Staubli VAL3: LasMAN.pjx

--- LasMAN.pjx ---
Parameters version=s7.7 stackSize=10000 millimeterUnit=true
Program file=Main.pgx
Program file=OnEvent1.pgx
Program file=OnEvent10.pgx
Program file=OnEvent11.pgx
Program file=OnEvent12.pgx
Program file=OnEvent13.pgx
Program file=OnEvent14.pgx
Program file=OnEvent15.pgx
Program file=OnEvent16.pgx
Program file=OnEvent17.pgx
Program file=OnEvent18.pgx
Program file=OnEvent19.pgx
Program file=OnEvent2.pgx
Program file=OnEvent3.pgx
Program file=OnEvent4.pgx
Program file=OnEvent5.pgx
Program file=OnEvent6.pgx
Program file=OnEvent7.pgx
Program file=OnEvent8.pgx
Program file=OnEvent9.pgx
Program file=Welcome.pgx
Program file=start.pgx
Program file=stop.pgx
Data file=LasMAN.dtx
Library alias=TxtFile path=Disk://TxtFile/TxtFile.pjx autoload=true password=
Library alias=UI path=Disk://StaubliUI/StaubliUI.pjx autoload=true password=
Library alias=DataBase path=Disk://DataBase/DataBase.pjx autoload=true password=
Library alias=Kit path=Disk://Kit/Kit.pjx autoload=true password=
Library alias=Teach path=Disk://Teach/Teach.pjx autoload=true password=
Library alias=IO path=Disk://IO/IO.pjx autoload=true password=
Library alias=ExtAxis path=Disk://extAxisCan/extAxisCan.pjx autoload=false password=

--- LasMAN.dtx ---
bool bExit
bool bSync
bool bWelcome = true

--- Main.pgx ---
program Main()
  local num l_nKey
begin

  //-----------------------------------------------------------------------
  //Header begin
  //Description of program
  //  根据不同类型的报警和当前机器人所处的运行状态处理报警事件
  //Input parameters
  //
  //Output paramaters
  //Example
  //  call Main()
  //History
  //  Creation : 2013-06-23
  //Header end
  //-----------------------------------------------------------------------
  //主程序


  //等按钮松开
  wait(getKey()==-1)
  do
    //每个操作模式之前的动作
    cls()
    userPage()
    resetMotion()
    call UI:Control_PanelMd("请等待，正在载入库......")


    //
    switch DataBase:nInterfaceType
      case 1
        //手动回零
        call OnEvent1()
      break
      case 2
        //手动对齐
        call OnEvent2()
      break
      case 3
        //编辑工艺
        call OnEvent3()
      break
      case 4
        //编辑动作
        call OnEvent4()
      break
      case 5
        //编辑产品
        call OnEvent5()
      break
      case 6
        //远程
        call OnEvent6()
      break
      //选项
      case 7
        call OnEvent7()
      break
      case 8
        //退出
        call OnEvent8()
      break
      case 9
        //主界面
        call OnEvent9()
      break
      case 10
        //示教产品的用户坐标系
        call OnEvent10()
      break

      case 11
        //示教产品偏差
        call OnEvent11()
      break

      //异步第七轴
      case 12
        call OnEvent12()
      break

      //生产
      case 13
        call OnEvent13()
      break


      //示教工具
      case 14
        call OnEvent14()
      break


      //示教Home
      case 15
        call OnEvent15()
      break


      //异步第八轴
      case 16
        call OnEvent16()
      break


      //替换空白调试文件
      case 17
        call OnEvent17()
      break


      //示教同步七轴
      case 18
        call OnEvent18()
      break

      //示教同步八轴
      case 19
        call OnEvent19()
      break


      //其他非法标志符，则退出
      default
        bExit=true
      break

    endSwitch

    delay(0)
  until bExit
  //Exit
  call stop()

end

--- start.pgx ---
program start()
  local bool l_bRes
begin

  //-----------------------------------------------------------------------
  //Header begin
  //Description of program
  //  LasMAN启动程序
  //Input parameters
  //
  //Output paramaters
  //
  //Creation : 2013.10.22 Ye yanjie  y.ye@staubli.com
  //Header end
  //-----------------------------------------------------------------------
  logMsg("运行lasman")
  DataBase:sSoftWareTime="2015_02_03"
  setTextMode(0)
  $jogPage(false)
  bWelcome=false
  taskCreate "Welcom",100,Welcome()



  //获取机器版本
  DataBase:sVersion[0]=getVersion("System")
  DataBase:sVersion[1]=getVersion("ArmType")
  DataBase:sVersion[2]=getVersion("Mounting")
  DataBase:sVersion[3]=getVersion("ControllerSN")
  DataBase:nRemoteProduct=0



  //删除备份
  $delete("Disk://BackUp")
  $delete("Disk://OffTxt")

  //参数初始化
  disablePower()
  bExit=false
  DataBase:nProductCount=0
  DataBase:bSaveTrajPoint=false
  TxtFile:tCfg.trsf=TxtFile:tFileTool.trsf={0,0,0,0,0,0}
  TxtFile:trPointCount={0,0,0,0,0,0}
  resetMotion()
  //设置默认的boxcar为0，10
  $setBoxcarFreq(0,10)


  //检查相应的文件是否正确
  call TxtFile:IsFileOK(l_bRes)
  if !l_bRes
    bWelcome=true
    delay(0)
    // popUpMsg("文本文件不正确!")
    call stop()
    return
  endIf

  //IO初始化
  call IO:Init()
  DataBase:nInterfaceType=9


  //外部轴初始化
  call Kit:ExtraSysAxisIni(l_bRes)
  if !l_bRes
    return
  endIf




  //建立新的进程
  taskCreate "LasMan",100,Main()
  taskCreate "Poll",100,Kit:Poll()
  bWelcome=true

end

--- OnEvent1.pgx ---
program OnEvent1()
  local bool l_bRes
begin
  //-----------------------------------------------------------------------
  //Header begin
  //LasMAN3.6
  //Description of program
  //
  //Input parameters
  //
  //Output paramaters
  //Example
  //  call OnEvent1()
  //History
  //  Creation : 2013-06-23  y.ye@staubli.com
  //Header end
  //-----------------------------------------------------------------------

  DataBase:bStopPoll=true
  call TxtFile:ReadCfg(l_bRes)
  IO:bWeldEnable=TxtFile:bWeldEnable
  IO:bWeldEnable=TxtFile:bWeldEnable
  IO:bExt7AxisEnable=TxtFile:b7Axis
  IO:bExt8AxisEnable=TxtFile:b8Axis
  DataBase:bStopPoll=false

  if l_bRes

    call Kit:GoHome()
  else
    popUpMsg("读取配置文件出错")
  endIf
  DataBase:nInterfaceType=9
end

--- OnEvent10.pgx ---
program OnEvent10()
begin
  //-----------------------------------------------------------------------
  //Header begin
  //LasMAN3.6
  //Description of program
  //
  //Input parameters
  //
  //Output paramaters
  //Example
  //  call OnEvent1()
  //History
  //  Creation : 2013-06-23  y.ye@staubli.com
  //Header end
  //-----------------------------------------------------------------------
  resetMotion()
  call Teach:TeachFrame(DataBase:fFrame)
  DataBase:nInterfaceType=9
end

--- OnEvent11.pgx ---
program OnEvent11()
begin
  //-----------------------------------------------------------------------
  //Header begin
  //LasMAN3.6
  //Description of program
  //
  //Input parameters
  //
  //Output paramaters
  //Example
  //  call OnEvent1()
  //History
  //  Creation : 2013-06-23  y.ye@staubli.com
  //Header end
  //-----------------------------------------------------------------------
  //示教偏差
  resetMotion()
  call Teach:TeachOffset(DataBase:fOffset)
  DataBase:nInterfaceType=9
end

--- OnEvent12.pgx ---
program OnEvent12()
begin
  //-----------------------------------------------------------------------
  //Header begin
  //LasMAN3.6
  //Description of program
  //
  //Input parameters
  //
  //Output paramaters
  //Example
  //  call OnEvent1()
  //History
  //  Creation : 2013-06-23  y.ye@staubli.com
  //Header end
  //-----------------------------------------------------------------------
  resetMotion()
  if TxtFile:b7Axis
    // call Teach:Teach7Axis(TxtFile:trAxisData.x,TxtFile:trAxisData.y,0)
    call Teach:TeachAxis(TxtFile:trAxisData.x,TxtFile:trAxisData.y,TxtFile:trAxisData.z,TxtFile:trAxisData.rx,false)
  else
    popUpMsg("请到选项界面中激活七轴")
  endIf
  DataBase:nInterfaceType=9
end

--- OnEvent13.pgx ---
program OnEvent13()
begin
  //-----------------------------------------------------------------------
  //Header begin
  //LasMAN3.6
  //Description of program
  //
  //Input parameters
  //
  //Output paramaters
  //Example
  //  call OnEvent1()
  //History
  //  Creation : 2013-06-23  y.ye@staubli.com
  //Header end
  //-----------------------------------------------------------------------
  resetMotion()
  call Teach:TeachProduct()
  DataBase:nInterfaceType=9
end

--- OnEvent14.pgx ---
program OnEvent14()
begin
  //-----------------------------------------------------------------------
  //Header begin
  //LasMAN3.6
  //Description of program
  //
  //Input parameters
  //
  //Output paramaters
  //Example
  //  call OnEvent1()
  //History
  //  Creation : 2013-06-23  y.ye@staubli.com
  //Header end
  //-----------------------------------------------------------------------
  resetMotion()
  call Teach:TeachTool()
  DataBase:nInterfaceType=9
end

--- OnEvent15.pgx ---
program OnEvent15()
begin
  //-----------------------------------------------------------------------
  //Header begin
  //LasMAN3.6
  //Description of program
  //
  //Input parameters
  //
  //Output paramaters
  //Example
  //  call OnEvent1()
  //History
  //  Creation : 2013-06-23  y.ye@staubli.com
  //Header end
  //-----------------------------------------------------------------------
  resetMotion()
  call Teach:TeachHome()
  DataBase:nInterfaceType=9
end

--- OnEvent16.pgx ---
program OnEvent16()
begin
  //-----------------------------------------------------------------------
  //Header begin
  //LasMAN3.6
  //Description of program
  //
  //Input parameters
  //
  //Output paramaters
  //Example
  //  call OnEvent1()
  //History
  //  Creation : 2013-06-23  y.ye@staubli.com
  //Header end
  //-----------------------------------------------------------------------
  resetMotion()
  if TxtFile:b8Axis
    // call Teach:Teach8Axis(TxtFile:trAxisData.rx,TxtFile:trAxisData.ry,0)
    call Teach:TeachAxis(TxtFile:trAxis8Data.x,TxtFile:trAxis8Data.y,TxtFile:trAxis8Data.z,TxtFile:trAxis8Data.rx,true)
  else
    popUpMsg("请到选项界面中激活八轴")
  endIf
  DataBase:nInterfaceType=9
end

--- OnEvent17.pgx ---
program OnEvent17()
  local bool l_bBool
begin
  //-----------------------------------------------------------------------
  //Header begin
  //LasMAN3.6
  //Description of program
  //
  //Input parameters
  //
  //Output paramaters
  //Example
  //  call OnEvent1()
  //History
  //  Creation : 2013-06-23  y.ye@staubli.com
  //Header end
  //-----------------------------------------------------------------------
  resetMotion()
  call UI:Control_YesNO("确定替换空白的调试文件吗?",l_bBool)
  if l_bBool
    call TxtFile:SaveNewProduct(l_bBool)

  endIf
  DataBase:nInterfaceType=9
end

--- OnEvent18.pgx ---
program OnEvent18()
  local bool l_bBool
begin
  //-----------------------------------------------------------------------
  //Header begin
  //LasMAN3.6
  //Description of program
  //
  //Input parameters
  //
  //Output paramaters
  //Example
  //  call OnEvent1()
  //History
  //  Creation : 2013-06-23  y.ye@staubli.com
  //Header end
  //-----------------------------------------------------------------------
  resetMotion()
  //      call UI:Control_YesNO("确定替换空白的调试文件吗?",l_bBool)
  //      if l_bBool
  //        call TxtFile:SaveNewProduct(l_bBool)
  //
  //      endIf
  call Teach:TeachSyncAxis()
  DataBase:nInterfaceType=9
end

--- OnEvent19.pgx ---
program OnEvent19()
  local bool l_bBool
begin
  //-----------------------------------------------------------------------
  //Header begin
  //LasMAN3.6
  //Description of program
  //
  //Input parameters
  //
  //Output paramaters
  //Example
  //  call OnEvent1()
  //History
  //  Creation : 2013-06-23  y.ye@staubli.com
  //Header end
  //-----------------------------------------------------------------------
  resetMotion()
  //      call UI:Control_YesNO("确定替换空白的调试文件吗?",l_bBool)
  //      if l_bBool
  //        call TxtFile:SaveNewProduct(l_bBool)
  //
  //      endIf

  call Teach:TeachSyncAxis()
  DataBase:nInterfaceType=9


end

--- OnEvent2.pgx ---
program OnEvent2()
  local bool l_bRes
begin
  //-----------------------------------------------------------------------
  //Header begin
  //LasMAN3.6
  //Description of program
  //
  //Input parameters
  //
  //Output paramaters
  //Example
  //  call OnEvent1()
  //History
  //  Creation : 2013-06-23  y.ye@staubli.com
  //Header end
  //-----------------------------------------------------------------------
  DataBase:bStopPoll=true
  call TxtFile:ReadCfg(l_bRes)
  IO:bWeldEnable=TxtFile:bWeldEnable
  DataBase:bStopPoll=false
  if l_bRes
    call Kit:Align(TxtFile:tCfg)
  else
    popUpMsg("读取配置文件出错")
  endIf
  DataBase:nInterfaceType=9
end

--- OnEvent3.pgx ---
program OnEvent3()
begin
  //-----------------------------------------------------------------------
  //Header begin
  //LasMAN3.6
  //Description of program
  //
  //Input parameters
  //
  //Output paramaters
  //Example
  //  call OnEvent1()
  //History
  //  Creation : 2013-06-23  y.ye@staubli.com
  //Header end
  //-----------------------------------------------------------------------

  call Teach:TeachPreset()
  DataBase:nInterfaceType=9
end

--- OnEvent4.pgx ---
program OnEvent4()
begin
  //-----------------------------------------------------------------------
  //Header begin
  //LasMAN3.6
  //Description of program
  //
  //Input parameters
  //
  //Output paramaters
  //Example
  //  call OnEvent1()
  //History
  //  Creation : 2013-06-23  y.ye@staubli.com
  //Header end
  //-----------------------------------------------------------------------

  call Teach:TeachAction()
  DataBase:nInterfaceType=9
end

--- OnEvent5.pgx ---
program OnEvent5()
begin
  //-----------------------------------------------------------------------
  //Header begin
  //LasMAN3.6
  //Description of program
  //
  //Input parameters
  //
  //Output paramaters
  //Example
  //  call OnEvent1()
  //History
  //  Creation : 2013-06-23  y.ye@staubli.com
  //Header end
  //-----------------------------------------------------------------------




  //单个七轴
  //2015.03.13
  //异步七轴
  if (TxtFile:b8Axis and DataBase:bSingleAxisMode)
    popUpMsg("异步外部轴配置出错")
    DataBase:nInterfaceType=9
    return
  endIf
  //**********


  if DataBase:bMutexAxis==false

  else
    //2014.4.15 为异步七八轴
    if (TxtFile:b7Axis or TxtFile:b8Axis) and DataBase:nWorkPlaceIndex<1
      // call UI:control_md
      call UI:Control_PanelMd("异步轴启动,等待工作台按钮信号")
      call UI:Control_BottomS(",,,,,,,终止")

      while DataBase:nWorkPlaceIndex<1
        if getKey()==278
          DataBase:nInterfaceType=9
          return
        endIf
        call IO:CanProduct(DataBase:nWorkPlaceIndex)
        delay(0)
      endWhile

    endIf

  endIf

  //2015.04.21
  TxtFile:trPointCount={0,0,0,0,0,0}
  call TxtFile:DeleteBuffTraj()



  //
  call Teach:TeachRecipe()
  DataBase:nInterfaceType=9


  //DataBase:sProductName=""
end

--- OnEvent6.pgx ---
program OnEvent6()
begin
  //-----------------------------------------------------------------------
  //Header begin
  //LasMAN3.6
  //Description of program
  //
  //Input parameters
  //
  //Output paramaters
  //Example
  //  call OnEvent1()
  //History
  //  Creation : 2013-06-23  y.ye@staubli.com
  //Header end
  //-----------------------------------------------------------------------
  if DataBase:nRemoteProduct==8888
    call Teach:TeachRemote()
  else
    popUpMsg("远程生产密码不正确")
  endIf
  DataBase:nInterfaceType=9
end

--- OnEvent7.pgx ---
program OnEvent7()
begin
  //-----------------------------------------------------------------------
  //Header begin
  //LasMAN3.6
  //Description of program
  //
  //Input parameters
  //
  //Output paramaters
  //Example
  //  call OnEvent1()
  //History
  //  Creation : 2013-06-23  y.ye@staubli.com
  //Header end
  //-----------------------------------------------------------------------

  call Teach:TeachConfig()
  DataBase:nInterfaceType=9
end

--- OnEvent8.pgx ---
program OnEvent8()
  local bool l_bRes
begin
  //-----------------------------------------------------------------------
  //Header begin
  //LasMAN3.6
  //Description of program
  //
  //Input parameters
  //
  //Output paramaters
  //Example
  //  call OnEvent1()
  //History
  //  Creation : 2013-06-23  y.ye@staubli.com
  //Header end
  //-----------------------------------------------------------------------

  call UI:Control_YesNO("确定要退出吗?",l_bRes)
  if l_bRes
    bExit=true
  else
    DataBase:nInterfaceType=9
  endIf

end

--- OnEvent9.pgx ---
program OnEvent9()
  local bool l_bBool
  local num l_nKey
begin
  //-----------------------------------------------------------------------
  //Header begin
  //LasMAN3.6
  //Description of program
  //
  //Input parameters
  //
  //Output paramaters
  //Example
  //  call OnEvent1()
  //History
  //  Creation : 2013-06-23  y.ye@staubli.com
  //Header end
  //-----------------------------------------------------------------------
  //初始化时所有的文件全部关闭
  //主界面也是安全界面
  resetMotion()
  //disablePower()
  call IO:SafteyIO()
  $fileClose(0)
  $fileClose(1)
  $fileClose(2)
  $fileClose(3)
  $fileClose(4)
  $fileClose(5)
  $fileClose(6)
  $fileClose(7)
  $fileClose(8)
  $fileClose(9)

  //设置MoveID为0
  setMoveId(0)
  //参数初始化
  DataBase:bSaveTrajPoint=false
  DataBase:bIOStart=false
  DataBase:bStopPoll=false
  DataBase:bUpload=false
  DataBase:bDebugMode=false
  TxtFile:cCfg.shoulder=ssame
  TxtFile:cCfg.elbow=esame
  TxtFile:cCfg.wrist=wsame
  DataBase:bMoveTask=false
  $jogContext(TxtFile:tCfg,world,0)
  DataBase:nSpeedPercent=1
  DataBase:nCycleCount=0
  DataBase:nWorkPlaceCount=0
  //强制一个按钮一次
  DataBase:nCycleMode=0
  DataBase:nWorkPlaceButto=-1
  DataBase:nWorkPlaceIndex=0
  DataBase:nPointType=0
  TxtFile:bReadProduct=false
  TxtFile:nReadCutCount=0
  DataBase:nProductIndex=0
  //2013.10.30
  //  for l_nKey=0 to size(DataBase:sProductName)-1
  //    DataBase:sProductName[l_nKey]=""
  //  endFor
  DataBase:nWpMutiCount[1]=DataBase:nWpMutiCount[2]=DataBase:nWpMutiCount[3]=DataBase:nWpMutiCount[4]=0
  //对数据强制进行初始化
  resize(TxtFile:pCut,1,1)
  resize(TxtFile:pMoveC,1,1)
  delay(0)
  resize(TxtFile:bMoveC,1,1)
  resize(TxtFile:trCut,1,1)

  TxtFile:pCut.config=TxtFile:pMoveC.config=TxtFile:cCfg



  //2014.11.28
  TxtFile:trPointCount={0,0,0,0,0,0}


  //安全化IO点
  call IO:SafteyIO()
  call IO:Light(1)

  //界面
  title("LasMAN3.6->主界面")
  if TxtFile:b7Axis
    call UI:Form_MainS("回零,七轴,工艺,动作,产品,远程,配置,退出")
  else
    call UI:Form_MainS("回零,对齐,工艺,动作,产品,远程,配置,退出")
  endIf
  gotoxy(1,11)
  if TxtFile:bWeldEnable
    put("激光精密焊接")
  else
    put("激光精密切割")
  endIf




  //事件响应
  while DataBase:nInterfaceType==9
    //
    //    if IO:dDio["In1_bHome"]==true
    //      DataBase:nInterfaceType=1
    //    endIf

    l_nKey=getKey()
    //按钮响应
    if l_nKey>=271 and l_nKey<=278
      if TxtFile:b7Axis and l_nKey==272
        DataBase:nInterfaceType=12
      else
        DataBase:nInterfaceType=l_nKey-270
      endIf
    endIf


    //使用默认的调试文件
    //double shift +Q
    if l_nKey==81
      DataBase:nInterfaceType=17
    endIf


    //示教Home
    if l_nKey==97
      DataBase:nInterfaceType=15
    endIf

    //示教TCP
    if l_nKey==122
      DataBase:nInterfaceType=14
    endIf

    //示教第七轴
    if l_nKey==119
      DataBase:nInterfaceType=12
    endIf


    //示教第八轴
    if l_nKey==115
      DataBase:nInterfaceType=16
    endIf

    //示教同步轴
    if l_nKey==120
      DataBase:nInterfaceType=18
    endIf


    //显示时间
    if l_nKey==-1
      gotoxy(20,9)

      if DataBase:bAlarm
        setTextMode(3)
        put("报警触发")
      else
        put("       ")
      endIf
      setTextMode(0)
      if TxtFile:b8Axis
        gotoxy(1,9)
        put("s->示教八轴")
      endIf

      gotoxy(20,11)
      put(left("时间:"+getDate("%H:%M:%S"),20))


      //同步七八轴
      //2014.07.30
      if TxtFile:bSync7Axis
        gotoxy(1,9)
        if !TxtFile:bSync8Axis
          put("同步七轴")
        else
          put("同步七八轴")
        endIf
      endIf


    endIf


    delay(0)
  endWhile

end

--- stop.pgx ---
program stop()
begin

  disablePower()
  resetMotion()
  $fileClose(0)
  $fileClose(1)
  $fileClose(2)
  $fileClose(3)
  $fileClose(4)
  $fileClose(5)
  $fileClose(6)
  $fileClose(7)
  $fileClose(8)
  $fileClose(9)
  if taskStatus("Poll")!=-1
    taskKill("Poll")
  endIf

  if taskStatus("SyncAxis")!=-1
    taskKill("SyncAxis")
  endIf
  //删除备份
  $delete("Disk://BackUp")
  $delete("Disk://OffTxt")

  call UI:Form_Bye()
  $jogPage(true)
  logMsg("关闭lasman")
end

--- Welcome.pgx ---
program Welcome()
begin

  call UI:Form_Welcome("激光软件LasMAN3.6",bWelcome)




end
